FUNCTION_BLOCK FB_TestHTTP_Get_openWeatherMapLat
VAR_INPUT
	bSend				: BOOL;
END_VAR
VAR_IN_OUT
	fbClient			: FB_IotHttpClient;
END_VAR
VAR_OUTPUT
	bBusy				: BOOL;
	bError				: BOOL;
END_VAR
VAR
	fbRequest			: FB_IotHttpRequest;
	fbJson				: FB_JsonDomParser;
	nState				: UDINT;
	RisingEdge			: R_TRIG;
	city : STRING;
	getweather : STRING := '/data/2.5/weather?q=';
	getweather2 : STRING := ',BE&appid=6E741a8faaaf146476fd94ab87413c7b&units=metric';
	getWeatherTotal : STRING(300);
	
	timerweather : ton;
	bGetContentResult	: BOOL;
	sContent			: STRING(511);	
	
	bGetJsonResult		: BOOL;
	jsonDoc				: SJsonValue;
	jsonVal				: SJsonValue;
	sResultValue		: STRING;
	
	nReqCount			: UDINT;	
	nResCount			: UDINT;
	nValidResCount		: UDINT;
	nErrCount			: UDINT;
	addstring: STRING;
	jsonprop: SJsonValue;
	jsonserial: SJsonValue;
	sTemp: LREAL ;
	
END_VAR

RisingEdge(CLK:= bSend);
IF autorefresh THEN 
	timerweather(in := NOT timerweather.Q, PT := T#30S);
END_IF


CASE nState OF
0:	
	IF RisingEdge.Q  THEN 
		addstring := concat(city , getweather2);
		getweathertotal := concat(getweather , addstring);
		
		
		IF fbRequest.SendRequest(sUri:= getweathertotal , fbClient:=fbClient, eRequestType:=ETcIotHttpRequestType.HTTP_Get, 0, 0, 0) THEN				
			nState:= 1;
			nReqCount:= nReqCount+1;
			bBusy:= TRUE;
			bError:= FALSE;
		END_IF					
	END_IF
	IF  timerweather.Q THEN 
		
		
		IF fbRequest.SendRequest(sUri:= getweathertotal , fbClient:=fbClient, eRequestType:=ETcIotHttpRequestType.HTTP_Get, 0, 0, 0) THEN				
			nState:= 1;
			nReqCount:= nReqCount+1;
			bBusy:= TRUE;
			bError:= FALSE;
		END_IF					
	END_IF
1:
	IF NOT fbRequest.bBusy THEN
		bError:= TRUE;
		IF NOT fbRequest.bError THEN				 
			bGetContentResult:= fbRequest.GetContent(pContent:= ADR(sContent), nContentSize:= SIZEOF(sContent), bSetNullTermination:= TRUE);
			IF fbRequest.nStatusCode >= 200 AND fbRequest.nStatusCode < 300 THEN
				bGetJsonResult:= FALSE;
				jsonDoc:= fbRequest.GetJsonDomContent(fbJson);
				IF jsonDoc <> 0 THEN
					parsen(); // do something with the weather data
					nValidResCount:= nValidResCount+1;
					bError:= FALSE;					
				END_IF							
				nResCount:= nResCount+1;			
			END_IF
		END_IF
		nState:= 0;
		bBusy:= FALSE;
		IF bError THEN
			nErrCount:= nErrCount+1;
		END_IF
	END_IF  	
END_CASE

ACTION parsen:
jsonprop := fbJson.FindMember(jsonDoc,'main');
IF (jsonprop <> 0) THEN
	jsonserial := fbjson.FindMember(jsonprop, 'temp');
	sTemp := fbjson.GetDouble(jsonserial);	
END_IF
END_ACTION

END_FUNCTION_BLOCK

(* stored: Version 1.1.0.1, ProductVersion 3.1.4024.9
   POU FB_TestHTTP_Get_openWeatherMapLat: Id {e991fc67-3d38-40ab-b2a0-bbe625e1fcff}, SpecialFunc None
   Action parsen: Id {38db57ef-ba31-4927-90d3-a9ba575e2786} *)
